TYPE ActionState :
STRUCT
	PreconditionsFullfilled	:	BOOL;
	IsActive	:	BOOL;
END_STRUCT
END_TYPE

(* stored: Version 1.1.0.1
   DUT ActionState: Id {9db9beef-3dc7-4065-befb-3aaed0f3090c} *)
